FUNCTION_BLOCK STRUCT_DEMUX (* Service Interface Function Block Type *)
  (* Standard: 61499-2; Description: Copyright (c) This program and the accompanying materials are made available under the terms of the Eclipse Public License 2.0 which is available at https://www.eclipse.org/legal/epl-2.0/ SPDX-License-Identifier: EPL-2.0 *)
  {SET_ATTRIBUTE(GenericClassName, 'GEN_STRUCT_DEMUX')}
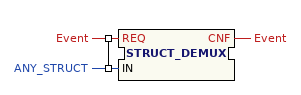
  EVENT_INPUT
    REQ WITH IN; (* Normal Execution Request *)
  END_EVENT
  EVENT_OUTPUT
    CNF; (* Execution Confirmation *)
  END_EVENT
  VAR_INPUT
    IN : ANY_STRUCT;
  END_VAR
  (* Service APPLICATION/RESOURCE: Service Interface Function Block Type *)
END_FUNCTION_BLOCK
